{attribute 'qualified_only'}
{attribute 'strict'}
{attribute 'to_string'}
TYPE LoadCellParameterizationSteps : (
    resetToFactorySettings := 0,
    setRatedOutput,
    setNominalLoad,
    setNominalOffset,
    setScalingFactor,
    Done
);
END_TYPE

(* stored: Version 1.1.0.1
   DUT LoadCellParameterizationSteps: Id {486860f9-ecfa-032a-01cb-e843f1b6f906} *)
